# B&R Automation Studio project TD52 (part 123)

#### general_HCCyclic.st
```iecst
(*******************************************************************************
general_HC		general functions

This code is confidential and proprietary to the INNIO Company.
It may not be used in any form, or reproduced in any manner,
without the express written permission of the INNIO Company.
Copyright, INNIO Company, 2019

Customized modifications: -
------------------------

History:
-------
V0.00.0	25.04.2012	lettenb.	new
V3.99.0 21.02.2013	lettenb.	cleanup
V4.03.0 11.01.2015	Denk		Bugfix, OUT_HC.tHWF_Dem.Do not implemented
		15.03.2016	Denk		Bugfix, Handbedienebene. OR IN_HC.tManAuxCtr.bHWF_Dem;
V4.05.0 11.12.2017	lettenb.	check para setup added
V4.14.0 08.11.2024	Bacci		OUT_HC.tECW_ShutOffVal_Dem.Do, OUT_HC.tValHeater_Dem.Do, OUT_HC.tFanRingHeater_Dem.Do added

Instructions for use:
--------------------
Outstandings:
------------
*******************************************************************************)

PROGRAM _INIT

	xECW_ShutOffVal_Dem_Active.enable := TRUE;
	xECW_ShutOffVal_Dem_Active.pPVstring := ADR('HalIO::ECW_ShutOffVal_Dem');
	xECW_ShutOffVal_Dem_Active();
	bECW_ShutOffVal_Dem_Exist := xECW_ShutOffVal_Dem_Active.exist;

	xValHeater_Dem_Active.enable := TRUE;
	xValHeater_Dem_Active.pPVstring := ADR('HalIO::ValHeater_Dem');
	xValHeater_Dem_Active();
	bValHeater_Dem_Exist := xValHeater_Dem_Active.exist;

	xFanRingHeater_Dem_Active.enable := TRUE;
	xFanRingHeater_Dem_Active.pPVstring := ADR('HalIO::FanRingHeater_Dem');
	xFanRingHeater_Dem_Active();
	bFanRingHeater_Dem_Exist := xFanRingHeater_Dem_Active.exist;

END_PROGRAM

PROGRAM _CYCLIC

	(* check para setup *)
	IN_HC.tPB2MM.bParaSetupOk;
	Para.iEng_Motortype;    (* MIN= 208   MAX= 920    *)
	Para.rN_EngStart_LimHi; (* MIN= 50.0  MAX= 2200.0 *)

	(* engine type defnition *)
	xEngType.Motortype := INT_TO_UINT(Para.iEng_Motortype);
	xEngType();

	(* engine operating mode selection *)
	bOMSS_Stop := FALSE;
	bOMSS_Man  := FALSE;
	bOMSS_Aut  := FALSE;
	bOMSS_Test := FALSE;
	bOMSS_Scav := FALSE;
	bOMSS_MAT  := FALSE;

	CASE IN_HC.iIdx_OMSS OF
	0:	bOMSS_Stop := TRUE;
	1:	bOMSS_Man  := TRUE;
		bOMSS_MAT  := TRUE;
	2:	bOMSS_Aut  := TRUE;
		bOMSS_MAT  := TRUE;
	3:	bOMSS_Test := TRUE;
		bOMSS_MAT  := TRUE;
	4:	bOMSS_Scav := TRUE;
	END_CASE;

	(* engine operating mode *)
	xOpMode(in:= IN_HC.iSt_OpMode);

	(*----------------------------------------------------------------------------------*)
	(* engine start speed *)
	xGR_MAXR_N_EngStart(In:= IN_HC.rN_EngAct, Gw:= Para.rN_EngStart_LimHi, Hy:= Para.rN_EngStart_HyHi);
	xTOF_N_EngStart(IN:= xGR_MAXR_N_EngStart.Q AND IN_HC.tPB2MM.bParaSetupOk, PT:= T#10s);
	bN_EngStart := xTOF_N_EngStart.Q;

	(*----------------------------------------------------------------------------------*)
	(* demand heating circuit flap *)
	OUT_HC.tHWF_Dem.Do := (IN_HC.bEng_Aux_Dem_CDR AND NOT IN_HC.bMsg1053 AND NOT IN_HC.bMsg1054 AND NOT IN_HC.bMsg1031)
						   OR IN_HC.tManAuxCtr.bHWF_Dem;

	(*----------------------------------------------------------------------------------*)
	(* demand 2-way shut off valve engine jacket water circuit (P.04(06)-YCS-029) *)
	OUT_HC.tECW_ShutOffVal_Dem.Do := IN_HC.bEng_Aux_Dem_CDR;

	(*----------------------------------------------------------------------------------*)
	(* demand 3-way valve heater (P.04/06/07-H-001) *)
	OUT_HC.tValHeater_Dem.Do := (NOT bT_AirOutdoor_Hi1 AND Para.bT_AirOutdoor_Active)
							 	 AND NOT IN_HC.bMsg1031
								 AND NOT IN_HC.bMsg1053
								 AND NOT IN_HC.bMsg1054;

	(*----------------------------------------------------------------------------------*)
	(* demand fan ring heater (P.04/06/07/09H-100) *)
	OUT_HC.tFanRingHeater_Dem.Do := (NOT bT_AirOutdoor_Hi1 AND Para.bT_AirOutdoor_Active)
							 		 AND NOT IN_HC.bMsg1031
									 AND NOT IN_HC.bMsg1053
									 AND NOT IN_HC.bMsg1054;

END_PROGRAM
```

#### general_HC.var
```iecst
VAR
	xGR_MAXR_N_EngStart : GR_MAXR;
	xTOF_N_EngStart : TOF;
	xECW_ShutOffVal_Dem_Active : OutExist;
	xValHeater_Dem_Active : OutExist;
	xFanRingHeater_Dem_Active : OutExist;
END_VAR
```

### Program Logical/HeatingCooling/BHV (IEC, version 4.11.0) - boiler house ventilation

#### BHVCyclic.st
```iecst
(*******************************************************************************
BHV	Boiler house ventilation

This code is confidential AND proprietary to the INNIO Company.
It may NOT be used in any form, or reproduced in any manner,
without the express written permission of the INNIO Company.
Copyright, INNIO Company, 2022

Customized modifications: -
------------------------

History:
-------
V4.03.0	25.07.2015	Plattner Johannes
V4.11.0	17.01.2022	lettenb.	bFail_BHV: tBHV_Dem.Do added to avoid warning at standstill, bugfix

Instructions FOR use:
--------------------

Boiler house ventilation, activation AND demand

Outstandings:
------------
*******************************************************************************)
PROGRAM _CYCLIC

	(* boiler house ventilation aktive*)
	(*----------------------------------------------------------------------------*)
	IF Para.bBHV_Active THEN

		OUT_HC.tBHV_Dem.Do	:= (IN_HC.tDemnd_BHV.Di AND NOT IN_HC.tManAuxCtr.bBHV_Dem_Man)
							   OR IN_HC.tManAuxCtr.bBHV_Dem;	(* Manual operating auxiliaries control - Handbedienebene *)
		bFail_BHV		:= NOT IN_HC.tBHV_Op.Di AND OUT_HC.tBHV_Dem.Do;
		(*----------------------------------------------------------------------------*)

		(* boiler house ventilation inaktive*)
		(*----------------------------------------------------------------------------*)
	ELSE

		OUT_HC.tBHV_Dem.Do	:= FALSE;
		bFail_BHV			:= FALSE;

	END_IF;
	(*----------------------------------------------------------------------------*)

END_PROGRAM
```

### Program Logical/HeatingCooling/Pr_ECW (IEC, version 4.12.0) - pressure engine cooling water

#### Pr_ECWCyclic.st
```iecst
(*******************************************************************************
Pr_ECW			pressure engine cooling water

This code is confidential and proprietary to the INNIO Company.
It may not be used in any form, or reproduced in any manner,
without the express written permission of the INNIO Company.
Copyright, INNIO Company, 2023

Customized modifications: -
------------------------

History:
-------
V0.1	20.10.1998	Pa			erstellt
 		24.11.1998	Pa			Korrekturlesung
V1.80	06.03.2003	LH			VISU-Grenzwerte erst aktiv wenn Rezepte auf Steuerung sind
 		18.03.2003	LH			Einlesen Analogeingang --> pb17
V2.06	01.07.2004	LH			Messignalstörung mit 2mA verzögert
V2.07	03.09.2004	LH			getrennte Verzögerungen für Messignalstörung eingeführt
V1.90	29.03.2004	LH			GW Kühlwasserdruck minimum warnend (Abstellung + 0,2bar)
 								GW Kühlwasserdruck maximum warnend (Abstellung - 0,4bar)
V2.20	24.04.2007	LH			Filter: 200ms --> 500ms (Hirzinger)
V2.50.0 28.01.2009	lettenb.	calm: GW_KDMI_W, HY_KDMI_W new parameter
V3.30.0	15.12.2011	lettenb.	GW_KDMA_W = GW_KDMA - 20 (war 40) (anforderung christian lang)
V3.99.0 21.02.2013	lettenb.	kwd -> Pr_ECW renamed, cleaning
V4.04.0	25.10.2016	lettenb.	measuring signal plausibility check (Functional Safety EN 13849)
		03.02.2017				bTON_EngRun added (validation just for 1 time)
		21.02.2017				2763: 0,1 -> 0,01 bar(acc.spec.thummer)
V4.05.0	22.12.2017	lettenb.	comment added: Safety-related application software source code (EN 13849-1 / 4.6.3)
		31.01.2018				2763 new logic(false alarms after long engine stand still time)(gfoeller)
V4.11.0	05.11.2021	Schmid		new Pr_ECW plausibility check logic
V4.12.0	28.03.2023	Perktold	variant mech Pump: Pr_ECW paus. check 10s longer monitoring, pressure limit 15mbar (former 20mbar)
V4.14.0 10.12.2024	Nagy		Added bPr_ECW_LoLoPrio2, bPr_ECW_HiHiPrio2 (2024-225)
Instructions for use:
--------------------

Outstandings:
------------
(*******************************************************************************)

PROGRAM _CYCLIC

(*---------------------------------------------------------------------------*)
	(* engine cooling water pressure *)

	(* low *)
	xGRMIN_Pr_ECW_Lo(In:= IN_HC.tPr_ECW.Ai, Gw:= Para.rPr_ECW_LimLo, Hy:= Para.rPr_ECW_HyLo);
    xTON_Pr_ECW_Lo(IN:= xGRMIN_Pr_ECW_Lo.Q AND IN_HC.tPB2MM.bParaSetupOk AND IN_HC.tPr_ECW.GoodQual, PT:= T#20s);
    bPr_ECW_Lo := xTON_Pr_ECW_Lo.Q;
	(* low during operation*)
	xGRMIN_Pr_ECW_LimOp(In:= IN_HC.tPr_ECW.Ai, Gw:= Para.rPr_ECW_LimLo_EngOp, Hy:= Para.rPr_ECW_HyLo);
	xTON_Pr_ECW_LimOp(IN:= xGRMIN_Pr_ECW_LimOp.Q AND IN_HC.tPB2MM.bParaSetupOk AND IN_HC.tPr_ECW.GoodQual, PT:= T#20s);
	bPr_ECW_LimOp := xTON_Pr_ECW_LimOp.Q;
	(********************************************************************************************************************
	Safety-related application software source code (EN 13849-1 / 4.6.3): BEGIN
	*********************************************************************************************************************)
	(* low low *)
	xGRMIN_Pr_ECW_LoLo(In:= IN_HC.tPr_ECW.Ai, Gw:= Para.rPr_ECW_LimLoLo, Hy:= Para.rPr_ECW_HyLoLo);
    xTON_Pr_ECW_LoLo(IN:= xGRMIN_Pr_ECW_LoLo.Q AND IN_HC.tPB2MM.bParaSetupOk AND IN_HC.tPr_ECW.GoodQual, PT:= T#3s);
    bPr_ECW_LoLo := xTON_Pr_ECW_LoLo.Q;
	(********************************************************************************************************************
	Safety-related application software source code (EN 13849-1 / 4.6.3): END
	*********************************************************************************************************************)
	(* low low Prio2 *)
	xGRMIN_Pr_ECW_LoLoPrio2(In:= IN_HC.tPr_ECW.Ai, Gw:= Para.rPr_ECW_LimLoLo - 0.2);
	xTON_Pr_ECW_LoLoPrio2(IN:= xGRMIN_Pr_ECW_LoLoPrio2.Q AND IN_HC.tPB2MM.bParaSetupOk AND IN_HC.tPr_ECW.GoodQual, PT:= T#3s);
	bPr_ECW_LoLoPrio2 := xTON_Pr_ECW_LoLoPrio2.Q;

	(* low 1 *)(* for custom use *)
	xGRMIN_Pr_ECW_Lo1(In:= IN_HC.tPr_ECW.Ai, Gw:= Para.rPr_ECW_LimLo1, Hy:= Para.rPr_ECW_HyLo1);
    xTON_Pr_ECW_Lo1(IN:= xGRMIN_Pr_ECW_Lo1.Q AND IN_HC.tPB2MM.bParaSetupOk, PT:= T#3s);
    OUT_HC.bPr_ECW_Lo1 := xTON_Pr_ECW_Lo1.Q;

	(* high *)
	xGRMAX_Pr_ECW_Hi(In:= IN_HC.tPr_ECW.Ai, Gw:= Para.rPr_ECW_LimHiHi - 0.20, Hy:= Para.rPr_ECW_HyHiHi);
    xTON_Pr_ECW_Hi(IN:= xGRMAX_Pr_ECW_Hi.Q AND IN_HC.tPB2MM.bParaSetupOk, PT:= T#10s);
	bPr_ECW_Hi := xTON_Pr_ECW_Hi.Q;

	(* high high *)
	xGRMAX_Pr_ECW_HiHi(In:= IN_HC.tPr_ECW.Ai, Gw:= Para.rPr_ECW_LimHiHi, Hy:= Para.rPr_ECW_HyHiHi);
    xTON_Pr_ECW_HiHi(IN:= xGRMAX_Pr_ECW_HiHi.Q AND IN_HC.tPB2MM.bParaSetupOk, PT:= T#10s);
	bPr_ECW_HiHi := xTON_Pr_ECW_HiHi.Q;

	(* high high Prio2 *)
	xGRMAX_Pr_ECW_HiHiPrio2(In:= IN_HC.tPr_ECW.Ai, Gw:= Para.rPr_ECW_LimHiHi + 0.2);
	bPr_ECW_HiHiPrio2 := xGRMAX_Pr_ECW_HiHiPrio2.Q AND IN_HC.tPB2MM.bParaSetupOk;

	(********************************************************************************************************************
	Safety-related application software source code (EN 13849-1 / 4.6.3): BEGIN
	*********************************************************************************************************************)
	(* measuring signal plausibility check - engine cooling water pressure (Functional Safety) *)

	(* reset saved pressure values *)
	IF xF_TRIG_Pcheck_Meas.Q THEN
		rPr_ECW_MaxValue		:=	0.0;
		rPr_ECW_MinValue		:=	100.0;
	END_IF;

	(* determine point when ECWP starts *)
	rN_ThresSpeedUp		:=	900.0;
	rN_ThresEngStop		:=	5.0;
	IF IN_HC.bECWP_MechDriven THEN	xR_TRIG_ECWP_start.CLK	:=	(IN_HC.rN_EngAct > rN_ThresEngStop);	// problem of failed start attempt!
	ELSE							xR_TRIG_ECWP_start.CLK	:=	IN_HC.tECWP1Dem.Do;
	END_IF;
	xR_TRIG_ECWP_start();
	xTP_Pr_ECW_Min_ECWP_start(IN:= xR_TRIG_ECWP_start.Q, PT:= T#10s);
	IF NOT IN_HC.tECWP1Dem.Do THEN	xTP_Pr_ECW_Min_ECWP_start(IN:= FALSE, PT:= T#0s);
	END_IF;

	(* define time window for tracking minimum ECW pressure *)
	xTON_NEng_Exc_Thres(IN := (IN_HC.rN_EngAct > rN_ThresSpeedUp), PT := T#10s);								//10s delay after speed up rpm reached before monitoring stop
	xRS_Pr_ECW_Min_Meas.SET		:=	xR_TRIG_ECWP_start.Q;
	IF IN_HC.bECWP_MechDriven THEN	xRS_Pr_ECW_Min_Meas.RESET1	:=	xTON_NEng_Exc_Thres.Q						// speed up rpm reached + 10s TON
																OR	(IN_HC.rN_EngAct < rN_ThresEngStop);		// interrupt with failed start attempt
	ELSE							xRS_Pr_ECW_Min_Meas.RESET1	:=	NOT xTP_Pr_ECW_Min_ECWP_start.Q;
	END_IF;
	xRS_Pr_ECW_Min_Meas();

	(* determine minimum ECW pressure during time window *)
	IF xRS_Pr_ECW_Min_Meas.Q1 THEN
		IF (IN_HC.tPr_ECW.Ai < rPr_ECW_MinValue) THEN	rPr_ECW_MinValue	:=	IN_HC.tPr_ECW.Ai;
		END_IF;
		IF (IN_HC.tPr_ECW.Ai > rPr_ECW_MaxValue) THEN	rPr_ECW_MaxValue	:=	IN_HC.tPr_ECW.Ai;
		END_IF;
	END_IF;

	(* mute plausibility check after ECWP operation *)
	IF IN_HC.bECWP_MechDriven THEN	xTOF_Pcheck_MonDeact.IN	:=	(IN_HC.rN_EngAct > rN_ThresEngStop);		// delay w.r.t. engine coming to standstill
	ELSE							xTOF_Pcheck_MonDeact.IN	:=	IN_HC.tECWP1Dem.Do;
	END_IF;
	xTOF_Pcheck_MonDeact(PT:= T#60s);
	bPcheck_Pr_ECW_MonRel	:=	NOT (xTOF_Pcheck_MonDeact.Q AND NOT xTOF_Pcheck_MonDeact.IN)	// mute for fast ECWP or engine restart
							AND	IN_HC.bEng_Aux_Dem												// check only active when engine/auxiliaries demanded
							AND	IN_HC.tPB2MM.bParaSetupOk;										// scaling parameters for Pr_ECW loaded

	(* trigger check evaluation *)
	xF_TRIG_Pcheck_Meas(CLK:= xRS_Pr_ECW_Min_Meas.Q1);

	IF xF_TRIG_Pcheck_Meas.Q AND bPcheck_Pr_ECW_MonRel THEN		bPr_ECW_PcheckFail	:=	((rPr_ECW_MaxValue - rPr_ECW_MinValue) < 0.015);
	ELSE														bPr_ECW_PcheckFail	:=	FALSE;
	END_IF;

	IF MM2VIS.bMsg2104 OR NOT IN_HC.tECWP_Op.Di THEN						bPr_ECW_PcheckFail := FALSE;
	ELSIF (rPr_ECW_MaxValue = 0.0) THEN										bPr_ECW_PcheckFail := FALSE; (* value not valid *)
	ELSIF (rPr_ECW_MinValue  = 0.0) OR (rPr_ECW_MinValue  = 100.0) THEN		bPr_ECW_PcheckFail := FALSE; (* value not valid *)
	END_IF;
	(********************************************************************************************************************
	Safety-related application software source code (EN 13849-1 / 4.6.3): END
	*********************************************************************************************************************)

END_PROGRAM
```

#### Pr_ECW.var
```iecst
VAR
	xGRMIN_Pr_ECW_Lo : GR_MINR;
	xTON_Pr_ECW_Lo : TON;
	xGRMIN_Pr_ECW_LimOp : GR_MINR;
	xTON_Pr_ECW_LimOp : TON;
	xGRMIN_Pr_ECW_LoLo : GR_MINR;
	xTON_Pr_ECW_LoLo : TON;
	xTON_Pr_ECW_LoLoPrio2 : TON;
	xGRMIN_Pr_ECW_LoLoPrio2 : GR_MINR;
	xGRMIN_Pr_ECW_Lo1 : GR_MINR;
	xTON_Pr_ECW_Lo1 : TON;
	xGRMAX_Pr_ECW_Hi : GR_MAXR;
	xTON_Pr_ECW_Hi : TON;
	xGRMAX_Pr_ECW_HiHi : GR_MAXR;
	xGRMAX_Pr_ECW_HiHiPrio2 : GR_MAXR;
	xTON_Pr_ECW_HiHi : TON;
	xR_TRIG_ECWP_start : R_TRIG; (*v4.11 new Pr_ECW plausibility check*)
	xTP_Pr_ECW_Min_ECWP_start : TP; (*v4.11new Pr_ECW plausibility check*)
	xTOF_Pcheck_MonDeact : TOF; (*v4.11new Pr_ECW plausibility check*)
	xRS_Pr_ECW_Min_Meas : RS; (*v4.11 new Pr_ECW plausibility check*)
	xF_TRIG_Pcheck_Meas : F_TRIG; (*v4.11 new Pr_ECW plausibility check*)
	rN_ThresSpeedUp : REAL; (*v4.11 new Pr_ECW plausibility check*)
	rN_ThresEngStop : REAL; (*v4.11 new Pr_ECW plausibility check*)
	bPcheck_Pr_ECW_MonRel : BOOL; (*v4.11 new Pr_ECW plausibility check*)
	rPr_ECW_MinValue : REAL := 100.0; (*v4.11 new Pr_ECW plausibility check*)
	rPr_ECW_MaxValue : REAL := 0.0; (*v4.11 new Pr_ECW plausibility check*)
	xTON_NEng_Exc_Thres : TON;
END_VAR
```

### Program Logical/HeatingCooling/T_CD (IEC, version 4.03.0) - temperature condensor circuit

#### T_CDCyclic.st
```iecst
(*******************************************************************************
T_CD		temperature condensor circuit

This code is confidential and proprietary to the INNIO Company.
It may not be used in any form, or reproduced in any manner,
without the express written permission of the INNIO Company.
Copyright, INNIO Company, 2019

Customized modifications: -
------------------------

History:
-------
V4.03.0	27.07.2015	Plattner	task created

Instructions for use:
--------------------

Outstandings:
------------
*******************************************************************************)

PROGRAM _CYCLIC
	(*-----------------------------------------------------------------------------*)
	(* condensor circuit supply temperature *)
	(* high *)
	xGRMAX_T_CD_Su_Hi(Gw:= Para.rT_CD_Su_LimHi, Hy:= Para.rT_CD_Su_HyHi, In:= IN_HC.tT_CD_Su.Ai);
	xTON_T_CD_Su_Hi(IN:= xGRMAX_T_CD_Su_Hi.Q AND IN_HC.tPB2MM.bParaSetupOk AND Para.bT_CD_Su_Active, PT:= T#2s);
	bT_CD_Su_Hi := xTON_T_CD_Su_Hi.Q;

	(*-----------------------------------------------------------------------------*)
	(* condensor circuit temperature *)
	(* high *)
	xGRMAX_T_CD_Re_Hi(In:= IN_HC.tT_CD_Re.Ai, Gw:= Para.rT_CD_Re_LimHi, Hy:= Para.rT_CD_Re_HyHi);
	xTON_T_CD_Re_Hi(IN := xGRMAX_T_CD_Re_Hi.Q AND IN_HC.tPB2MM.bParaSetupOk AND Para.bT_CD_Re_Active, PT := T#2s);
	bT_CD_Re_Hi := xTON_T_CD_Re_Hi.Q;

	(*-----------------------------------------------------------------------------*)

END_PROGRAM
```

#### T_CD.var
```iecst
VAR
	xTON_T_CD_Su_Hi : TON;
	xGRMAX_T_CD_Su_Hi : GR_MAXR;
	xGRMAX_T_CD_Re_Hi : GR_MAXR;
	xTON_T_CD_Re_Hi : TON;
END_VAR
```

### Program Logical/HeatingCooling/T_ECW (IEC, version 4.00.0) - temperature engine cooling water

#### T_ECWCyclic.st
```iecst
(*******************************************************************************
T_ECW			temperature engine cooling water

This code is confidential and proprietary to the INNIO Company.
It may not be used in any form, or reproduced in any manner,
without the express written permission of the INNIO Company.
Copyright, INNIO Company, 2019

Customized modifications: -
------------------------

History:
-------
V0.1	01.10.1998	Pa			erstellt
		24.11.1998	Pa			korrekturlesung
V170	03.04.2002	LH			Verzögerung Kühlwassertemperatur max. => 5min
								Grenzwert Kühlwassertemperatur max. + 2°C (Abstellung)
V180	06.03.2003	LH			VISU-Grenzwerte erst aktiv wenn Rezepte auf Steuerung sind
		18.03.2003	LH			Einlesen Analogeingang --> pb17
V3.99.0	20.02.2013	lettenb.	kwtp renamed T_ECW, cleaning
								new param.for cooling water bypass valve
V4.00.0 19.03.2015				xGRMIN_T_ECW_Lo: avoid bMsg1145 at cold restart within hysteresis

Instructions for use:
--------------------

Outstandings:
------------
(*******************************************************************************)

PROGRAM _CYCLIC

(*---------------------------------------------------------------------------*)
	(* engine cooling water temperature *)

	(* low *)
	IF IN_HC.tPB2MM.bParaSetupOk THEN (* avoid bMsg1145 at cold restart within hysteresis *)
		 xGRMIN_T_ECW_Lo(In:= IN_HC.tT_ECW.Ai, Gw:= Para.rT_ECW_LimLo, Hy:= Para.rT_ECW_HyLo);
	ELSE xGRMIN_T_ECW_Lo(In:= 1.0, Gw:= 0.0, Hy:= 0.0);
	END_IF;
	xTON_T_ECW_Lo(IN:= xGRMIN_T_ECW_Lo.Q AND IN_HC.tPB2MM.bParaSetupOk, PT:= T#2s);
    OUT_HC.bT_ECW_Lo := xTON_T_ECW_Lo.Q;

	(*high preheating off *)
	xGRMAX_T_ECW_PreH_OFF(In:= IN_HC.tT_ECW.Ai, Gw:= Para.rT_ECW_PreH_LimOFF, Hy:= Para.rT_ECW_PreH_HyOFF);
    xTON_T_ECW_PreH_OFF(IN:= xGRMAX_T_ECW_PreH_OFF.Q AND IN_HC.tPB2MM.bParaSetupOk, PT:= T#2s);
    OUT_HC.bT_ECW_PreH_OFF := xTON_T_ECW_PreH_OFF.Q;

	(* high synch/load release *)
	xGRMAX_T_ECW_RelLoad(In:= IN_HC.tT_ECW.Ai, Gw:= Para.rT_ECW_LimRelLoad, Hy:= Para.rT_ECW_HyRelLoad);
    xTON_T_ECW_RelLoad(IN:= xGRMAX_T_ECW_RelLoad.Q AND IN_HC.tPB2MM.bParaSetupOk, PT:= T#2s);
    OUT_HC.bT_ECW_RelLoad := xTON_T_ECW_RelLoad.Q;

	(* high *)
	xGRMAX_T_ECW_Hi(In:= IN_HC.tT_ECW.Ai, Gw:= Para.rT_ECW_LimHi, Hy:= Para.rT_ECW_HyHi);
    xTON_T_ECW_Hi(IN:= xGRMAX_T_ECW_Hi.Q AND IN_HC.tPB2MM.bParaSetupOk, PT:= T#300s);
    OUT_HC.bT_ECW_Hi := xTON_T_ECW_Hi.Q;

	(* high high *)
	xGRMAX_T_ECW_HiHi(In:= IN_HC.tT_ECW.Ai, Gw:= Para.rT_ECW_LimHi + 2.0, Hy:= Para.rT_ECW_HyHi);
    xTON_T_ECW_HiHi(IN:= xGRMAX_T_ECW_HiHi.Q AND IN_HC.tPB2MM.bParaSetupOk, PT:= T#2s);
    bT_ECW_HiHi := xTON_T_ECW_HiHi.Q;

	(* high P2 *)
	xGRMAX_T_ECW_HiHiPrio2(In:= IN_HC.tT_ECW.Ai, Gw:= Para.rT_ECW_LimHi + 5.0, Hy:= Para.rT_ECW_HyHi);
	xTON_T_ECW_HiHiPrio2(IN:= xGRMAX_T_ECW_HiHiPrio2.Q AND IN_HC.tPB2MM.bParaSetupOk, PT:= T#2s);
	bT_ECW_HiHiPrio2 := xTON_T_ECW_HiHiPrio2.Q;

	(* high 1 *)
	xGRMAX_T_ECW_Hi1(In:= IN_HC.tT_ECW.Ai, Gw:= Para.rT_ECW_LimHi1, Hy:= Para.rT_ECW_HyHi1);
    xTON_T_ECW_Hi1(IN:= xGRMAX_T_ECW_Hi1.Q AND IN_HC.tPB2MM.bParaSetupOk, PT:= T#2s);
    bT_ECW_Hi1 := xTON_T_ECW_Hi1.Q;

	(* high 2 *)
	xGRMAX_T_ECW_Hi2(In:= IN_HC.tT_ECW.Ai, Gw:= Para.rT_ECW_LimHi2, Hy:= Para.rT_ECW_HyHi2);
    xTON_T_ECW_Hi2(IN:= xGRMAX_T_ECW_Hi2.Q AND IN_HC.tPB2MM.bParaSetupOk, PT:= T#2s);
    bT_ECW_Hi2 := xTON_T_ECW_Hi2.Q;

	(*---------------------------------------------------------------------------*)
	(* engine cooling water temperature - bypass valve *)
	xGRMIN_T_ECW_BpV(In:= IN_HC.tT_ECW.Ai, Gw:= Para.rT_ECW_LimBpV, Hy:= Para.rT_ECW_HyBpV);
	xTON_T_ECW_BpV(IN:= xGRMIN_T_ECW_BpV.Q, PT:= T#2s);

	bECW_DemBpV := (	IN_HC.bEng_Aux_Dem AND xTON_T_ECW_BpV.Q)
    			OR (NOT IN_HC.bEng_Aux_Dem AND IN_HC.bEng_Aux_Dem_CDR);
    OUT_HC.tECW_DemBpV.Do 	:= bECW_DemBpV;

	(*---------------------------------------------------------------------------*)
	(*	engine cooling water bypass pump *)
    bECW_DemBpP 			:= bECW_DemBpV;
    OUT_HC.tECW_DemBpP.Do 	:= bECW_DemBpP;

(*---------------------------------------------------------------------------*)

END_PROGRAM
```

#### T_ECW.var
```iecst
VAR
	xGRMIN_T_ECW_Lo : GR_MINR;
	xTON_T_ECW_Lo : TON;
	xGRMAX_T_ECW_PreH_OFF : GR_MAXR;
	xTON_T_ECW_PreH_OFF : TON;
	xGRMAX_T_ECW_RelLoad : GR_MAXR;
	xTON_T_ECW_RelLoad : TON;
	xGRMAX_T_ECW_Hi : GR_MAXR;
	xTON_T_ECW_Hi : TON;
	xGRMAX_T_ECW_HiHi : GR_MAXR;
	xTON_T_ECW_HiHi : TON;
	xGRMAX_T_ECW_HiHiPrio2 : GR_MAXR;
	xTON_T_ECW_HiHiPrio2 : TON;
	xGRMAX_T_ECW_Hi1 : GR_MAXR;
	xTON_T_ECW_Hi1 : TON;
	xGRMAX_T_ECW_Hi2 : GR_MAXR;
	xTON_T_ECW_Hi2 : TON;
	xGRMIN_T_ECW_BpV : GR_MINR;
	xTON_T_ECW_BpV : TON;
END_VAR
```

### Program Logical/HeatingCooling/T_EO (IEC, version 3.99.0) - temperature engine oil

#### T_EOCyclic.st
```iecst
(*******************************************************************************
T_EO			engine oil temperature

This code is confidential and proprietary to the INNIO Company.
It may not be used in any form, or reproduced in any manner,
without the express written permission of the INNIO Company.
Copyright, INNIO Company, 2019

Customized modifications: -
------------------------

History:
-------
V3.99.0	20.02.2013	lettenb.	new from task: otp

Instructions for use:
--------------------

Outstandings:
------------
(*******************************************************************************)

PROGRAM _CYCLIC

	(* engine oil temperature high 1 *)
	xGR_MAXR_T_EO_Hi1(In:= IN_HC.tT_EO.Ai, Gw:= Para.rT_EO_LimHi1, Hy:= Para.rT_EO_HyHi1);
	xTON_T_EO_Hi1(IN:= xGR_MAXR_T_EO_Hi1.Q AND IN_HC.tPB2MM.bParaSetupOk, PT:= T#2s);
	bT_EO_Hi1 := xTON_T_EO_Hi1.Q;

	(* engine oil temperature high 2 *)
	xGR_MAXR_T_EO_Hi2(In:= IN_HC.tT_EO.Ai, Gw:= Para.rT_EO_LimHi2, Hy:= Para.rT_EO_HyHi2);
	xTON_T_EO_Hi2(IN:= xGR_MAXR_T_EO_Hi2.Q AND IN_HC.tPB2MM.bParaSetupOk, PT:= T#2s);
	bT_EO_Hi2 := xTON_T_EO_Hi2.Q;

END_PROGRAM
```

#### T_EO.var
```iecst
VAR
	xTON_T_EO_Hi1 : TON;
	xGR_MAXR_T_EO_Hi1 : GR_MAXR;
	xTON_T_EO_Hi2 : TON;
	xGR_MAXR_T_EO_Hi2 : GR_MAXR;
END_VAR
```

### Program Logical/HeatingCooling/T_HW (IEC, version 4.05.0) - temperature heat water

#### T_HWCyclic.st
```iecst
(*******************************************************************************
T_HW		temperature heat water

This code is confidential and proprietary to the INNIO Company.
It may not be used in any form, or reproduced in any manner,
without the express written permission of the INNIO Company.
Copyright, INNIO Company, 2019

Customized modifications: -
------------------------

History:
-------
V3.99.0	20.02.2013	lettenb.	from task vltp, rltp, rltp_nk, rlt_m
								p_limitHC included
		14.03.2012	lettenb.	p_lim --> p_red (power red.from act.frozen power value) request: systems/thummer mathias
V4.00.0	01.07.2014	lettenb.	bT_HW_Su_Hi/HiHi: AND Para.bT_HW_Su_Active added, bugfix
V4.03.0	29.07.2015	plattner	heat circuit temperature added
V4.04.0 29.07.2016	lettenb.	2nd bT_HW_ReBeEng_Hi building removed, cleanup
		12.09.2016				comment removed
V4.05.0 13.06.2017	lettenb.	rP_Red_T_ECW_Low_Norm added, SWAT920/3

Instructions for use:
--------------------

Outstandings:
------------
*******************************************************************************)

PROGRAM _CYCLIC
	(*-----------------------------------------------------------------------------*)
	(* heat water supply temperature *)
	(* high *) (* W2430 *)
	xGRMAX_T_HW_Su_Hi(Gw:= Para.rT_HW_Su_LimHi, Hy:= Para.rT_HW_Su_HyHi, In:= IN_HC.tT_HW_Su.Ai);
	xTON_T_HW_Su_Hi(IN:= xGRMAX_T_HW_Su_Hi.Q AND IN_HC.tPB2MM.bParaSetupOk AND Para.bT_HW_Su_Active, PT:= T#2s);
	bT_HW_Su_Hi := xTON_T_HW_Su_Hi.Q;

	(* high high *) (* A1063 *)
	xGRMAX_T_HW_Su_HiHi(Gw:= Para.rT_HW_Su_LimHiHi, Hy:= Para.rT_HW_Su_HyHiHi, In:= IN_HC.tT_HW_Su.Ai);
	xTON_T_HW_Su_HiHi(IN := xGRMAX_T_HW_Su_HiHi.Q AND IN_HC.tPB2MM.bParaSetupOk AND Para.bT_HW_Su_Active, PT := T#2s);
	bT_HW_Su_HiHi := xTON_T_HW_Su_HiHi.Q;

	(*-----------------------------------------------------------------------------*)
	(* heat water return temperature *)
	(* high *)
	xGRMAX_T_HW_Re_Hi(In:= IN_HC.tT_HW_Re.Ai, Gw:= Para.rT_HW_Re_LimHi, Hy:= Para.rT_HW_Re_HyHi);
	xTON_T_HW_Re_Hi(IN := xGRMAX_T_HW_Re_Hi.Q AND IN_HC.tPB2MM.bParaSetupOk AND Para.bT_HW_Re_Active, PT := T#2s);
	bT_HW_Re_Hi := xTON_T_HW_Re_Hi.Q;

	(* high high *)
	xGRMAX_T_HW_Re_HiHi(In := IN_HC.tT_HW_Re.Ai, Gw := Para.rT_HW_Re_LimHiHi, Hy := Para.rT_HW_Re_HyHiHi);
	xTON_T_HW_Re_HiHi(IN:= xGRMAX_T_HW_Re_HiHi.Q AND IN_HC.tPB2MM.bParaSetupOk AND Para.bT_HW_Re_Active, PT:= T#2s);
	bT_HW_Re_HiHi := xTON_T_HW_Re_HiHi.Q;

	(*-----------------------------------------------------------------------------*)
	(* heat water return temperature after emergency cooler *)
	(* high *)
	xGRMAX_T_HW_ReAfEC_Hi(In:= IN_HC.tT_HW_ReAfEC.Ai, Gw:= Para.rT_HW_ReAfEC_LimHi, Hy:= Para.rT_HW_ReAfEC_HyHi);
	xTON_T_HW_ReAfEC_Hi(IN:= xGRMAX_T_HW_ReAfEC_Hi.Q AND IN_HC.tPB2MM.bParaSetupOk, PT:= T#2s);
	bT_HW_ReAfEC_Hi := xTON_T_HW_ReAfEC_Hi.Q;

	(* high high *)
	xGRMAX_T_HW_ReAfEC_HiHi(In:= IN_HC.tT_HW_ReAfEC.Ai, Gw:= Para.rT_HW_ReAfEC_LimHiHi, Hy:= Para.rT_HW_ReAfEC_HyHiHi);
	xTON_T_HW_ReAfEC_HiHi(IN:= xGRMAX_T_HW_ReAfEC_HiHi.Q AND IN_HC.tPB2MM.bParaSetupOk, PT:= T#2s);
	bT_HW_ReAfEC_HiHi := xTON_T_HW_ReAfEC_HiHi.Q;

	(*-----------------------------------------------------------------------------*)
	(* heat water return temperature before engine *)
	(* high *)
	xGRMAX_T_HW_ReBeEng_Hi(In:= IN_HC.tT_HW_ReBeEng.Ai, Gw:= Para.rT_HW_ReBeEng_LimHi, Hy:= Para.rT_HW_ReBeEng_HyHi, );
	xTON_T_HW_ReBeEng_Hi(IN:= xGRMAX_T_HW_ReBeEng_Hi.Q AND IN_HC.tPB2MM.bParaSetupOk, PT:= T#2s);
	bT_HW_ReBeEng_Hi := xTON_T_HW_ReBeEng_Hi.Q;

	(* high high *)(* reserve *)
	xGRMAX_T_HW_ReBeEng_HiHi(In:= IN_HC.tT_HW_ReBeEng.Ai, Gw:= Para.rT_HW_ReBeEng_LimHiHi, Hy:= Para.rT_HW_ReBeEng_HyHiHi, );
	xTON_T_HW_ReBeEng_HiHi(IN:= xGRMAX_T_HW_ReBeEng_HiHi.Q AND IN_HC.tPB2MM.bParaSetupOk, PT:= T#2s);
	bT_HW_ReBeEng_HiHi := xTON_T_HW_ReBeEng_HiHi.Q;

	(*-----------------------------------------------------------------------------*)
	(* heat circuit temperature *)
	(* high *)
	xGRMAX_T_HW_HC_Re_Hi(Gw:= Para.rT_HW_HC_Re_LimHi, Hy:= Para.rT_HW_HC_Re_HyHi, In:= IN_HC.tT_HW_HC_Re.Ai);
	xTON_T_HW_HC_Re_Hi(IN:= xGRMAX_T_HW_HC_Re_Hi.Q AND IN_HC.tPB2MM.bParaSetupOk AND Para.bT_HW_HC_Re_Active, PT:= T#2s);
	bT_HW_HC_Re_Hi := xTON_T_HW_HC_Re_Hi.Q;

	(*-----------------------------------------------------------------------------*)
	(* power reduction by heat water return temperature high *)
	(* selection *)
	CASE Para.iPred_T_HW_Re_Sel OF
		0:	rT_HW_Re := 0;						(* disabled	*)
		1:	rT_HW_Re := IN_HC.tT_HW_Re.Ai;		(* P.06(04)-TI-012	(NUT12) *)
		2:	rT_HW_Re := IN_HC.tT_HW_ReAfEC.Ai;	(* P.06(04)-TI-015	(NUT15) *)
		3:	rT_HW_Re := IN_HC.tT_HW_ReBeEng.Ai;	(* M.06(04)-TI-001	(NUT56) *)
		ELSE
			rT_HW_Re :=0;
	END_CASE;

	IF rT_HW_Re <= Para.rT_Pred_HW_Re_Start THEN
		rP_Act_Norm_frozen := IN_HC.rP_Act_Norm_Filt;
	END_IF;

	IF Para.iPred_T_HW_Re_Sel <> 0 AND rT_HW_Re > Para.rT_Pred_HW_Re_Start THEN
		OUT_HC.rP_Red_T_HWR_Norm := LIMIT(0.5, rP_Act_Norm_frozen - ((rT_HW_Re - Para.rT_Pred_HW_Re_Start) * Para.rPred_T_HW_Re_Rate), 1.0);
	ELSE
		OUT_HC.rP_Red_T_HWR_Norm := 1.0;
	END_IF;

	(* power reduction by engine cooling water return temperature low - warm up operation *)
	IF IN_HC.tT_ECW.Ai < Para.rT_ECW_PwrRamp_LimLo AND bOMSS_Man AND xEngType.Type9 THEN
		OUT_HC.rP_Red_T_ECW_Low_Norm := 0.40;//%Pnom(10MW) = ca.4MW
	ELSE
		OUT_HC.rP_Red_T_ECW_Low_Norm := 1.0;
	END_IF;

	(* power reduction by engine cooling water temperature high *)
	OUT_HC.rP_Red_T_ECW_Norm := LIMIT(0.5, 1.0 - ((IN_HC.tT_ECW.Ai - Para.rT_Pred_ECW_Start) * Para.rPred_ECW_Rate), 1.0);

	(*-----------------------------------------------------------------------------*)

	(*-----------------------------------------------------------------------------*)

END_PROGRAM
```

#### T_HW.var
```iecst
VAR
	xGRMAX_T_HW_Su_Hi : GR_MAXR;
	xTON_T_HW_Su_Hi : TON;
	xGRMAX_T_HW_Su_HiHi : GR_MAXR;
	xTON_T_HW_Su_HiHi : TON;
	xGRMAX_T_HW_Re_Hi : GR_MAXR;
	xTON_T_HW_Re_Hi : TON;
	xGRMAX_T_HW_Re_HiHi : GR_MAXR;
	xTON_T_HW_Re_HiHi : TON;
	xGRMAX_T_HW_ReBeEng_Hi : GR_MAXR;
	xTON_T_HW_ReBeEng_Hi : TON;
	xGRMAX_T_HW_ReBeEng_HiHi : GR_MAXR;
	xTON_T_HW_ReBeEng_HiHi : TON;
	xGRMAX_T_HW_ReAfEC_Hi : GR_MAXR;
	xTON_T_HW_ReAfEC_Hi : TON;
	xGRMAX_T_HW_ReAfEC_HiHi : GR_MAXR;
	xTON_T_HW_ReAfEC_HiHi : TON;
	rT_HW_Re : REAL;
	rP_Act_Norm_frozen : REAL;
	xGRMAX_T_HW_HC_Re_Hi : GR_MAXR;
	xTON_T_HW_HC_Re_Hi : TON;
END_VAR
```

### Program Logical/HeatingCooling/T_AirOutdoor (IEC, version 3.99.0) - temperature air outdoor

#### T_AirOutdoor.st
```iecst
(*******************************************************************************
T_AirOutdoor		temperature air outdoor

This code is confidential and proprietary to the INNIO Company.
It may not be used in any form, or reproduced in any manner,
without the express written permission of the INNIO Company.
Copyright, INNIO Company, 2019

Customized modifications: -
------------------------

History:
-------
V2.10	18.05.2004	LH			erstellt
V3.99.0	21.02.2013	lettenb.	ult --> T_AirOutdoor renamed

Instructions for use:
--------------------

Outstandings:
------------
*******************************************************************************)

PROGRAM _CYCLIC

	(* outdoor air temperature *)

	(* high 1 *)
	xGRMAX_T_AirOutdoor_Hi1(In:= IN_HC.tT_AirOutdoor.Ai, Gw:= Para.rT_AirOutdoor_LimHi1, Hy:= Para.rT_AirOutdoor_HyHi1);
	bT_AirOutdoor_Hi1 := IN_HC.tPB2MM.bParaSetupOk AND xGRMAX_T_AirOutdoor_Hi1.Q AND Para.bT_AirOutdoor_Active;

	(* high 2 *)
	xGRMAX_T_AirOutdoor_Hi2(In:= IN_HC.tT_AirOutdoor.Ai, Gw:= Para.rT_AirOutdoor_LimHi2, Hy:= Para.rT_AirOutdoor_HyHi2);
	bT_AirOutdoor_Hi2 := IN_HC.tPB2MM.bParaSetupOk AND xGRMAX_T_AirOutdoor_Hi2.Q AND Para.bT_AirOutdoor_Active;

	(* high 3 *)
	xGRMAX_T_AirOutdoor_Hi3(In:= IN_HC.tT_AirOutdoor.Ai, Gw:= Para.rT_AirOutdoor_LimHi3, Hy:= Para.rT_AirOutdoor_HyHi3);
	bT_AirOutdoor_Hi3 := IN_HC.tPB2MM.bParaSetupOk AND xGRMAX_T_AirOutdoor_Hi3.Q AND Para.bT_AirOutdoor_Active;

	(* high 4 *)
	xGRMAX_T_AirOutdoor_Hi4(In:= IN_HC.tT_AirOutdoor.Ai, Gw:= Para.rT_AirOutdoor_LimHi4, Hy:= Para.rT_AirOutdoor_HyHi4);
	bT_AirOutdoor_Hi4 := IN_HC.tPB2MM.bParaSetupOk AND xGRMAX_T_AirOutdoor_Hi4.Q AND Para.bT_AirOutdoor_Active;

END_PROGRAM
```

#### T_AirOutdoor.var
```iecst
VAR
	xGRMAX_T_AirOutdoor_Hi1 : GR_MAXR;
	xGRMAX_T_AirOutdoor_Hi2 : GR_MAXR;
	xGRMAX_T_AirOutdoor_Hi3 : GR_MAXR;
	xGRMAX_T_AirOutdoor_Hi4 : GR_MAXR;
END_VAR
```

### Program Logical/HeatingCooling/T_Ch (IEC, version 4.07.0) - temperature charge air/mixture

#### T_ChCyclic.st
```iecst
(*******************************************************************************
T_Ch 		temperature charge air/mixture

This code is confidential and proprietary to the INNIO Company.
It may not be used in any form, or reproduced in any manner,
without the express written permission of the INNIO Company.
Copyright, INNIO Company, 2019

Customized modifications: -
------------------------

History:
-------
V3.99.0	21.02.2013	lettenb.	new for MM_HC
V4.07.0	09.08.2018	Schmid		2nd low temperature charge cooling circuit added

Instructions for use:
--------------------

Outstandings:
------------
*******************************************************************************)

PROGRAM _CYCLIC

	(* charge temperature t2' *)
	(* high 1 *)
	xGRMAX_T_Ch_Hi1(In:= IN_HC.rT_Ch_T2s_Avg, Gw:= Para.rT_Ch_LimHi1, Hy:= Para.rT_Ch_HyHi1);
	bT_Ch_Hi1 := xGRMAX_T_Ch_Hi1.Q AND IN_HC.tPB2MM.bParaSetupOk;

	(* high 2 *)
	xGRMAX_T_Ch_Hi2(In:= IN_HC.rT_Ch_T2s_Avg, Gw:= Para.rT_Ch_LimHi2, Hy:= Para.rT_Ch_HyHi2);
	bT_Ch_Hi2 := xGRMAX_T_Ch_Hi2.Q AND IN_HC.tPB2MM.bParaSetupOk;

	(* charge temperature before high-pressure turbo charger T1-HP - 2nd LT cooling circuit*)
	(* high 1 *)
	xGRMAX_T_Ch_T1HP_Hi1(In:= IN_HC.rT_Ch_T1HP_Avg, Gw:= Para.rT_Ch_T1HP_LimHi1, Hy:= Para.rT_Ch_T1HP_HyHi1);
	bT_Ch2_Hi1 := xGRMAX_T_Ch_T1HP_Hi1.Q AND IN_HC.tPB2MM.bParaSetupOk;

	(* high 2 *)
	xGRMAX_T_Ch_T1HP_Hi2(In:= IN_HC.rT_Ch_T1HP_Avg, Gw:= Para.rT_Ch_T1HP_LimHi2, Hy:= Para.rT_Ch_T1HP_HyHi2);
	bT_Ch2_Hi2 := xGRMAX_T_Ch_T1HP_Hi2.Q AND IN_HC.tPB2MM.bParaSetupOk;

END_PROGRAM
```

#### T_Ch.var
```iecst
VAR
	xGRMAX_T_Ch_Hi1 : GR_MAXR;
	xGRMAX_T_Ch_Hi2 : GR_MAXR;
	xGRMAX_T_Ch_T1HP_Hi1 : GR_MAXR;
	xGRMAX_T_Ch_T1HP_Hi2 : GR_MAXR;
END_VAR
```

### Program Logical/HeatingCooling/EC_Seq (IEC, version 4.03.0) - emergency cooler sequence

#### EC_SeqCyclic.st
```iecst
(*******************************************************************************
EC_Seq 			emergency cooler - sequence for 16 stages

This code is confidential and proprietary to the INNIO Company.
It may not be used in any form, or reproduced in any manner,
without written permission of the INNIO Company.
Copyright, INNIO Company, 2019

Customized modifications: -
------------------------

History:
-------
V0.1 	31-01-2003	Thaler		generated
     	21-03-2003	Thaler		last modification
V1.81	16-06-2003	LH			bits für Anzeige auf VISU
V1.82	16-09-2003	LH			Variable für XT-Anzeige
V2.07.1a31-03-2005	LH			Variable für Freigabe XT-Anzeige
V2.30	24-01-2008	LH			Variable für Freigabe XT-Anzeige gelöscht (Parameter!)
V3.99.0	21.02.2013	lettenb.	kv_seq -> EC_Seq renamed
V4.03.0 07.08.2015  Denk		Manual operating auxiliaries control functionality added

Instructions for use:
--------------------

Outstandings:
------------
*******************************************************************************)
PROGRAM _CYCLIC

	(* Manual operating auxiliaries control - Handbedienebene *)
	K_Var := LIMIT(0, Para.iEC_OpMode, 3);
	FOR i:= 1 TO Para.iEC_NumStages BY 1 DO
		IF 	(K_Var > 0 AND K_Var < 4) THEN
			K_ST1_ManAuxCtr  := IN_HC.tManAuxCtr.bEC_DemFan;
			K_ST2_ManAuxCtr  :=	IN_HC.tManAuxCtr.bEC_DemFan;
			K_ST3_ManAuxCtr  :=	IN_HC.tManAuxCtr.bEC_DemFan;
			K_ST4_ManAuxCtr  := IN_HC.tManAuxCtr.bEC_DemFan;
			K_ST5_ManAuxCtr  := IN_HC.tManAuxCtr.bEC_DemFan;
			K_ST6_ManAuxCtr  := IN_HC.tManAuxCtr.bEC_DemFan;
			K_ST7_ManAuxCtr  := IN_HC.tManAuxCtr.bEC_DemFan;
			K_ST8_ManAuxCtr  := IN_HC.tManAuxCtr.bEC_DemFan;
			K_ST9_ManAuxCtr  := IN_HC.tManAuxCtr.bEC_DemFan;
			K_ST10_ManAuxCtr := IN_HC.tManAuxCtr.bEC_DemFan;
			K_ST11_ManAuxCtr := IN_HC.tManAuxCtr.bEC_DemFan;
			K_ST12_ManAuxCtr := IN_HC.tManAuxCtr.bEC_DemFan;
			K_ST13_ManAuxCtr := IN_HC.tManAuxCtr.bEC_DemFan;
			K_ST14_ManAuxCtr := IN_HC.tManAuxCtr.bEC_DemFan;
			K_ST15_ManAuxCtr := IN_HC.tManAuxCtr.bEC_DemFan;
			K_ST16_ManAuxCtr := IN_HC.tManAuxCtr.bEC_DemFan;

			IF IN_HC.tManAuxCtr.bEC_DemFan = TRUE THEN
				iSumEC_Stages_ManAuxCtr := Para.iEC_NumStages;
			ELSE
				iSumEC_Stages_ManAuxCtr := 0;
			END_IF;
		END_IF;
	END_FOR;

	(* connection of in-/outputs *)
	EN[1]  := K_ST_1;
	EN[2]  := K_ST_2;
	EN[3]  := K_ST_3;
	EN[4]  := K_ST_4;
	EN[5]  := K_ST_5;
	EN[6]  := K_ST_6;
	EN[7]  := K_ST_7;
	EN[8]  := K_ST_8;
	EN[9]  := K_ST_9;
	EN[10] := K_ST_10;
	EN[11] := K_ST_11;
	EN[12] := K_ST_12;
	EN[13] := K_ST_13;
	EN[14] := K_ST_14;
	EN[15] := K_ST_15;
	EN[16] := K_ST_16;

	IN[1]  := K_ST1;
	IN[2]  := K_ST2;
	IN[3]  := K_ST3;
	IN[4]  := K_ST4;
	IN[5]  := K_ST5;
	IN[6]  := K_ST6;
	IN[7]  := K_ST7;
	IN[8]  := K_ST8;
	IN[9]  := K_ST9;
	IN[10] := K_ST10;
	IN[11] := K_ST11;
	IN[12] := K_ST12;
	IN[13] := K_ST13;
	IN[14] := K_ST14;
	IN[15] := K_ST15;
	IN[16] := K_ST16;

	OUT_HC.tEC_DemFan1.Do := Q[1] OR K_ST1_ManAuxCtr;
	OUT_HC.tEC_DemFan2.Do := Q[2] OR K_ST2_ManAuxCtr;
	OUT_HC.tEC_DemFan3.Do := Q[3] OR K_ST3_ManAuxCtr;
	OUT_HC.tEC_DemFan4.Do := Q[4] OR K_ST4_ManAuxCtr;
	OUT_HC.tEC_DemFan5.Do := Q[5] OR K_ST5_ManAuxCtr;
	OUT_HC.tEC_DemFan6.Do := Q[6] OR K_ST6_ManAuxCtr;
	OUT_HC.tEC_DemFan7.Do := Q[7] OR K_ST7_ManAuxCtr;
	OUT_HC.tEC_DemFan8.Do := Q[8] OR K_ST8_ManAuxCtr;
	OUT_HC.tEC_DemFan9.Do := Q[9] OR K_ST9_ManAuxCtr;
	OUT_HC.tEC_DemFan10.Do := Q[10] OR K_ST10_ManAuxCtr;
	OUT_HC.tEC_DemFan11.Do := Q[11] OR K_ST11_ManAuxCtr;
	OUT_HC.tEC_DemFan12.Do := Q[12] OR K_ST12_ManAuxCtr;
	OUT_HC.tEC_DemFan13.Do := Q[13] OR K_ST13_ManAuxCtr;
	OUT_HC.tEC_DemFan14.Do := Q[14] OR K_ST14_ManAuxCtr;
	OUT_HC.tEC_DemFan15.Do := Q[15] OR K_ST15_ManAuxCtr;
	OUT_HC.tEC_DemFan16.Do := Q[16] OR K_ST16_ManAuxCtr;

	(******************************************************************************)

	and_16b   (ADR(EN), ADR(Q), ADR(Q));	(* switch off "Q" if "EN" is FALSE:	"Q" := "EN" AND "Q" *)
	andnt_16b (ADR(EN), ADR(Q), ADR(RDY));	(* enabled outputs with status FALSE: "RDY" := "EN" AND NOT "Q" *)

	(* SEQU_C = stage number for stage numbers > iPriorityStage *)
	FOR i := (iPriorityStage + 1) TO 16 BY 1 DO
		SEQU_C[i] := i;
	END_FOR;

	(* SEQU_C = stage number + 100 for stage numbers <= iPriorityStage *)
	FOR i := iPriorityStage TO 1 BY -1 DO
		 SEQU_C[i] := i + 100;
	END_FOR;

	min_16di (ADR(RDY), ADR(SEQU_C), ADR(NEXT_ON));	(* stage for next on  as BOOL *)
	min_16di (ADR(Q), ADR(SEQU_C), ADR(NEXT_OFF)); 	(* stage for next off as BOOL *)

	iNextOn   := max_i_16b (ADR(NEXT_ON)); 			(* stage for next on  as INT  *)
	iNextOff  := max_i_16b (ADR(NEXT_OFF));			(* stage for next off as INT  *)

	iIN := max_i_16b (ADR(IN));						(* input : number of stages as INT *)
	iQ  := sum_16b (ADR(Q));   						(* output: number of stages as INT *)

	IF (iIN > iQ) THEN
		Q[iNextOn] := TRUE;
		iPriorityStage := iNextOn;
	END_IF;

	IF (iIN < iQ) THEN
		Q[iNextOff] := FALSE;
	END_IF;

	(******************************************************************************)

	(* bits for visu *)
	summe := 0;
	FOR i:= 1 TO 16 BY 1 DO
		summe := summe + Q[i];
	END_FOR;

	K_byte1	:= FALSE;
	K_byte2	:= FALSE;

	K_bit10	:= FALSE;
	K_bit11	:= FALSE;
	K_bit12	:= FALSE;

	K_bit20	:= FALSE;
	K_bit21	:= FALSE;
	K_bit22	:= FALSE;

	IF	(summe > 0) AND (summe < 9) THEN
		K_byte1	:= TRUE;
	END_IF;

	IF	((summe = 2) OR (summe = 4) OR (summe = 6) OR (summe = 8)) THEN
		K_bit10	:= TRUE;
	END_IF;

	IF	((summe = 3) OR (summe = 4) OR (summe = 7) OR (summe = 8)) THEN
		K_bit11	:= TRUE;
	END_IF;

	IF	((summe = 5) OR (summe = 6) OR (summe = 7) OR (summe = 8)) THEN
		K_bit12	:= TRUE;
	END_IF;

	IF	(summe > 8) THEN
		K_byte2	:= TRUE;
	END_IF;

	IF	((summe = 10) OR (summe = 12) OR (summe = 14) OR (summe = 16)) THEN
		K_bit20	:= TRUE;
	END_IF;

	IF	((summe = 11) OR (summe = 12) OR (summe = 15) OR (summe = 16)) THEN
		K_bit21	:= TRUE;
	END_IF;

	IF	((summe = 13) OR (summe = 14) OR (summe = 15) OR (summe = 16)) THEN
		K_bit22	:= TRUE;
	END_IF;

	IF iSumEC_Stages_ManAuxCtr > 0 THEN
		iSumEC_Stages := iSumEC_Stages_ManAuxCtr; 	(* Manual operating auxiliaries control - Handbedienebene to vis *)
	ELSE
		iSumEC_Stages := summe;						(* to vis *)
	END_IF;

END_PROGRAM
```

#### EC_Seq.var
```iecst
VAR
	K_bit10 : BOOL := 0; (* Kühlerstufe 1-8 bit0 *)
	K_bit11 : BOOL := 0; (* Kühlerstufe 1-8 bit1 *)
	K_bit12 : BOOL := 0; (* Kühlerstufe 1-8 bit2 *)
	K_bit20 : BOOL := 0; (* Kühlerstufe 9-16 bit0 *)
	K_bit21 : BOOL := 0; (* Kühlerstufe 9-16 bit1 *)
	K_bit22 : BOOL := 0; (* Kühlerstufe 9-16 bit2 *)
	K_byte1 : BOOL := 0; (* Kühlerstufen 1-8 *)
	K_byte2 : BOOL := 0; (* Kühlerstufen 9-16 *)
	IN : ARRAY[0..16] OF BOOL;
	Q : ARRAY[0..16] OF BOOL;
	RDY : ARRAY[0..16] OF BOOL;
	EN : ARRAY[0..16] OF BOOL;
	iQ : INT;
	iIN : INT;
	iPriorityStage : INT;
	SEQU_C : ARRAY[0..16] OF DINT;
	NEXT_ON : ARRAY[0..16] OF BOOL;
	NEXT_OFF : ARRAY[0..16] OF BOOL;
	i : INT;
	iNextOn : INT;
	iNextOff : INT;
	summe : USINT := 0;
	K_Var : INT; (*emergency cooler variant*)
	iSumEC_Stages_ManAuxCtr : INT; (*summary emergency cooler stages from Manual operating auxiliaries control *)
END_VAR
```

### Program Logical/HeatingCooling/EC (IEC, version 4.10.0) - emergency cooler

#### ECCyclic.st
```iecst
(*******************************************************************************
EC 			emergency cooler

This code is confidential and proprietary to the INNIO Company.
It may not be used in any form, or reproduced in any manner,
without written permission of the INNIO Company.
Copyright, INNIO Company, 2021

Customized modifications: -
------------------------

History:
-------
V0.1	03.07.1998	Pa			erstellt
 		24.11.1998	Pa			korrekturlesung
V172	20.08.2002	LH			überarbeitet
V173	27.09.2002	LH			Fehler in Abschaltung Stufe 7 korrigiert
V180	25.02.2003	LH			nkv_schr --> kv_schr, Ausgangsvariablen umbenannt, Grenzwerte über Rezept
		07.03.2003	LH			Freigabe Kühler umgebaut für Service
V181	05.06.2003	LH			Kontaktplan --> strukturierten Text
V183	16.09.2003	LH			Korrektur Vorzeichen P-Anteil
		12.12.2003	LH			Variante Kombikühler
V2071	03.01.2005	LH			Korrektur Start Kühler durch Temperaturgrenzwerte,
								Ansteuerung Notkühlpumpe nur über Ventilstellung
V2071b	28.06.2005	LH			Korrektur Start Kühler über Ventilstellung
V190	08.09.2004	LH			Erweiterung auf 11 Regler für XT
V2102	22.11.2006	LH			Korrektur Ansteuerung Notkühlpumpe für ausgebundenen Notkühlkreis und Kombikühler
V230	24.01.2008	LH			Abarbeitung nur wenn Kühler vorhanden ist (Para.iEC_OpMode <> 0)
		06.02.2008	LH			angepasst an Auto-Tune Regler
V2.34.0 23.10.2008	lettenb.	OUT_HC.bEC_Stage1-16:(FA_K_EIN.Q OR Kombi_K) added(fan only if OUT_HC.bEC_DemP)
V3.10.0 17.02.2010	lettenb. 	corr.demand fan stage 1,2 (brackets)	fehlerbehebung(robert mayer)
V3.20.0	11.11.2010	lettenb. 	Anz_anfhbt, K_Var, K_Anz, K_reg -> parameters
V3.99.0	21.02.2013	lettenb.	parts from pb3 included
		24.06.2013				GRMin_Ventpos2,xGRMax_Ventpos2,GRMax_Ventpos4: Hy:= 1->0.01, bugfix
V4.00.0	03.03.2015	lettenb.	K_frg (IN_HC.bEC_Rel) moved to MM_CU
V4.03.0 07.08.2015  Denk		Manual operating auxiliaries control functionality added
V4.07.0	08.01.2019	Schmid		redundant pump control
V4.10.0	02.02.2021	lettenb.	OUT_HC.tEC_DemPump.Do only when	auxiliaries demanded(bEng_Aux_Dem_CDR)
								for safety purposes: otherwise pump starts immediately when y-limit is reached(or setted manually)
								OUT_HC.bEmCWP_Dem for K_Var > 0 prepared for reduntant pumps, bugfix

Instructions for use:
--------------------

Outstandings:
------------
(*******************************************************************************)
PROGRAM _CYCLIC

	(*------------------------------------------------------------------------------------------*)
	(* parameters *)
	K_Var 		:= 				LIMIT(0, Para.iEC_OpMode, 3);			(* cooler type
																			0 = cooler simple version
																			1 = cooler level dependent on valve position
																			2 = cooler level dependent on temperature
																			3 = combined cooler (type 1 and 2) *)
	K_Anz 		:= INT_TO_USINT(LIMIT(1, Para.iEC_NumStages, 16));		(* number cooler stages *)
	Anz_anfhbt	:= INT_TO_USINT(LIMIT(0, Para.iEC_NumDemAux, K_Anz));	(* number cooler stages with demand auxiliaries *)
	K_reg		:= INT_TO_USINT(LIMIT(1, Para.iEC_NumCtr, 11));			(* number controller for y *)
	K_nmp		:= 						 Para.bEC_St1onlyP;				(* selection first stage without fan (only pump)*)
																		(* only IF setting FOR number cooler stages with demand auxiliaries = 0 ! *)
																		(* this option reduces effective cooler fan stages by 1 step ! *)

	(*------------------------------------------------------------------------------------------*)
	(* release emergency cooler from monitoring (from MM_CU) *)
	IN_HC.bEC_Rel;

	(*------------------------------------------------------------------------------------------*)
	(* release for external cooler *)
	OUT_HC.tExCo_Rel.Do	:=	IN_HC.bEng_Aux_Dem_CDR
						AND(bT_HW_Re_Hi OR bT_HW_ReBeEng_Hi);

	(*==========================================================================================*)
	(* emergency cooler control - simple version *)
	IF K_Var = 0 THEN

		OUT_HC.tEC_DemPump.Do	:= (IN_HC.bEC_Rel
								AND IN_HC.bEng_Aux_Dem_CDR AND (bT_AirOutdoor_Hi1 OR NOT Para.bT_AirOutdoor_Active))
								OR IN_HC.tManAuxCtr.bEC_DemPump;	(* Manual operating auxiliaries control - Handbedienebene *)
		OUT_HC.bEmCWP_Dem		:= OUT_HC.tEC_DemPump.Do;

		(* stage 1 *)
		K_ST1	:=  IN_HC.bEC_Rel
				AND	IN_HC.bEng_Aux_Dem_CDR
				AND(bT_AirOutdoor_Hi1 OR NOT Para.bT_AirOutdoor_Active);

		(* stage 2 *)
		K_ST2	:=	IN_HC.bEC_Rel
				AND K_ST1
				AND	IN_HC.bEng_Aux_Dem_CDR
				AND(bT_AirOutdoor_Hi2 OR NOT Para.bT_AirOutdoor_Active);

		(* stage 3 *)
		K_ST3	:=	IN_HC.bEC_Rel
				AND K_ST2
				AND((IN_HC.bEng_Aux_Dem_CDR AND bT_AirOutdoor_Hi3) OR (bT_ECW_Hi1 AND NOT Para.bT_AirOutdoor_Active));

		(* stage 4 *)
		K_ST4	:=	IN_HC.bEC_Rel
				AND K_ST3
				AND((IN_HC.bEng_Aux_Dem_CDR AND bT_AirOutdoor_Hi4) OR (bT_ECW_Hi2 AND NOT Para.bT_AirOutdoor_Active));

	END_IF;

	(*==========================================================================================*)
	(* emergency cooler control - stepper version *)

	IF K_Var > 0 THEN
	(* cooler stages ON/OFF (cooler type 2/3)*)
		bEC_Up   :=     bT_ECW_Hi2 OR      bT_Ch_Hi2 OR      bT_EO_Hi2;
		bEC_Down := NOT bT_ECW_Hi1 AND NOT bT_Ch_Hi1 AND NOT bT_EO_Hi1;

		(*---------------------------------------------------------------------------------------*)
		FA_INIT_0.Word	:=	INT_TO_UINT(K_Var);
		FA_INIT_0;
		K_vent			:=	FA_INIT_0.Bit00;
		K_temp			:=	FA_INIT_0.Bit01;
		muell			:=	FA_INIT_0.Bit02;
		muell			:=	FA_INIT_0.Bit03;
		muell			:=	FA_INIT_0.Bit04;
		muell			:=	FA_INIT_0.Bit05;
		muell			:=	FA_INIT_0.Bit06;
		muell			:=	FA_INIT_0.Bit07;
		muell			:=	FA_INIT_0.Bit08;
		muell			:=	FA_INIT_0.Bit09;
		muell			:=	FA_INIT_0.Bit10;
		muell			:=	FA_INIT_0.Bit11;
		muell			:=	FA_INIT_0.Bit12;
		muell			:=	FA_INIT_0.Bit13;
		muell			:=	FA_INIT_0.Bit14;
		muell			:=	FA_INIT_0.Bit15;

		IF	K_vent AND K_temp	THEN
			Kombi_K		:=	1;
		ELSE
			Kombi_K		:=	0;
		END_IF;

		IF	Anz_anfhbt > 0	THEN
			K_nmp		:=	0;
			K_anfhbt	:=	1;
		ELSE
			K_anfhbt	:=	0;
		END_IF;

		FOR	i			:=	1 TO 16 BY 1 DO
			anfhbt[i]	:=	0;
		END_FOR;
		FOR	i			:=	1 TO Anz_anfhbt BY 1 DO
			anfhbt[i]	:=	1;
		END_FOR;

		(* number effective cooler stages *)
		Anz_st			:=	MIN(K_Anz - (MAX(Anz_anfhbt, 1) - 1) + BOOL_TO_USINT(K_nmp), 16);

		zw				:=	1;
		FOR i			:=	1 TO Anz_st BY 1	DO
			zw			:=	zw * 2;
		END_FOR;

		FA_INIT_1.Word	:=	UDINT_TO_UINT(zw - 1);
		FA_INIT_1;
		ST_1			:=	FA_INIT_1.Bit00;
		ST_2			:=	FA_INIT_1.Bit01;
		ST_3			:=	FA_INIT_1.Bit02;
		ST_4			:=	FA_INIT_1.Bit03;
		ST_5			:=	FA_INIT_1.Bit04;
		ST_6			:=	FA_INIT_1.Bit05;
		ST_7			:=	FA_INIT_1.Bit06;
		ST_8			:=	FA_INIT_1.Bit07;
		ST_9			:=	FA_INIT_1.Bit08;
		ST_10			:=	FA_INIT_1.Bit09;
		ST_11			:=	FA_INIT_1.Bit10;
		ST_12			:=	FA_INIT_1.Bit11;
		ST_13			:=	FA_INIT_1.Bit12;
		ST_14			:=	FA_INIT_1.Bit13;
		ST_15			:=	FA_INIT_1.Bit14;
		ST_16			:=	FA_INIT_1.Bit15;

		(* activation cooler stages *)
		Anz_vent		:=	MIN(K_Anz, 16 - BOOL_TO_USINT(K_nmp));

		zw				:=	1;
		FOR	i			:=	1 TO Anz_vent BY 1	DO
			zw			:=	zw * 2;
		END_FOR;

		FA_INIT_2.Word	:=	UDINT_TO_UINT(zw - 1);
		FA_INIT_2;
		K_ST_1			:=	FA_INIT_2.Bit00;
		K_ST_2			:=	FA_INIT_2.Bit01;
		K_ST_3			:=	FA_INIT_2.Bit02;
		K_ST_4			:=	FA_INIT_2.Bit03;
		K_ST_5			:=	FA_INIT_2.Bit04;
		K_ST_6			:=	FA_INIT_2.Bit05;
		K_ST_7			:=	FA_INIT_2.Bit06;
		K_ST_8			:=	FA_INIT_2.Bit07;
		K_ST_9			:=	FA_INIT_2.Bit08;
		K_ST_10			:=	FA_INIT_2.Bit09;
		K_ST_11			:=	FA_INIT_2.Bit10;
		K_ST_12			:=	FA_INIT_2.Bit11;
		K_ST_13			:=	FA_INIT_2.Bit12;
		K_ST_14			:=	FA_INIT_2.Bit13;
		K_ST_15			:=	FA_INIT_2.Bit14;
		K_ST_16			:=	FA_INIT_2.Bit15;

		(* 3-way cooler valve *)
		CASE K_reg OF							(* selection plant ctr # for 3-way valve (1-11) (cooler type 1/3) *)
		1:	F_SPSR		:=	IN_HC.tCtr_Cust1_In.enable;	(* 1-8 = custom plant ctr - device temperature *)
			rValvePos	:=	IN_HC.tCtr_Cust1_Out.Y;
			REG_INVERT	:=	Para.tCtr_Cust1.invert;
		2:	F_SPSR		:=	IN_HC.tCtr_Cust2_In.enable;
			rValvePos	:=	IN_HC.tCtr_Cust2_Out.Y;
			REG_INVERT	:=	Para.tCtr_Cust2.invert;
		3:	F_SPSR		:=	IN_HC.tCtr_Cust3_In.enable;
			rValvePos	:=	IN_HC.tCtr_Cust3_Out.Y;
			REG_INVERT	:=	Para.tCtr_Cust3.invert;
		4:	F_SPSR		:=	IN_HC.tCtr_Cust4_In.enable;
			rValvePos	:=	IN_HC.tCtr_Cust4_Out.Y;
			REG_INVERT	:=	Para.tCtr_Cust4.invert;
		5:	F_SPSR		:=	IN_HC.tCtr_Cust5_In.enable;
			rValvePos	:=	IN_HC.tCtr_Cust5_Out.Y;
			REG_INVERT	:=	Para.tCtr_Cust5.invert;
		6:	F_SPSR		:=	IN_HC.tCtr_Cust6_In.enable;
			rValvePos	:=	IN_HC.tCtr_Cust6_Out.Y;
			REG_INVERT	:=	Para.tCtr_Cust6.invert;
		7:	F_SPSR		:=	IN_HC.tCtr_Cust7_In.enable;
			rValvePos	:=	IN_HC.tCtr_Cust7_Out.Y;
			REG_INVERT	:=	Para.tCtr_Cust7.invert;
		8:	F_SPSR		:=	IN_HC.tCtr_Cust8_In.enable;
			rValvePos	:=	IN_HC.tCtr_Cust8_Out.Y;
			REG_INVERT	:=	Para.tCtr_Cust8.invert;
		9:	F_SPSR		:=	tCtr_ChC_In.enable;			(* 9   = charge temperature controller *)
			rValvePos	:=	tCtr_ChC_Out.Y;
			REG_INVERT	:=	Para.tCtr_ChC.invert;
		10:	F_SPSR		:=	tCtr_HWRe_In.enable;		(* 10  =  heat water return temperature controller *)
			rValvePos	:=	tCtr_HWRe_Out.Y;
			REG_INVERT	:=	Para.tCtr_HWRe.invert;
		11:	F_SPSR		:=	tCtr_EC_In.enable;			(* 11  =  heat water return temperature after cooler controller *)
			rValvePos	:=	tCtr_EC_Out.Y;
			REG_INVERT	:=	Para.tCtr_EC.invert;
		ELSE
			F_SPSR		:=	FALSE;
			rValvePos	:=	0.0;
			REG_INVERT	:=	FALSE;
		END_CASE;

		IF	NOT REG_INVERT	THEN
			rValvePos	:=	1.0 - rValvePos;
		END_IF;

	    (*---------------------------------------------------------------------------*)
		(* cooler ON *)
		xGRMax_Ventpos5(Gw:= Para.rEC_ValPosLimHi_On, Hy:= Para.rEC_ValPosHyHi_On, In:= rValvePos);

	    (*---------------------------------------------------------------------------*)
		xTOF_K_AUS.IN	:= (K_vent AND xGRMax_Ventpos5.Q AND IN_HC.tPB2MM.bParaSetupOk AND USINT_TO_BOOL(F_SPSR))
						OR (K_temp AND ((bEC_Up OR K_EIN AND NOT bEC_Down) OR K_EIN AND M_KV2));
		xTOF_K_AUS.PT	:=	Para.tiEC_DelayOff;
		xTOF_K_AUS;

		K_EIN			:=	(xTOF_K_AUS.Q OR K_anfhbt) AND IN_HC.bEng_Aux_Dem_CDR AND IN_HC.bEC_Rel;

	    (*---------------------------------------------------------------------------*)
		(* cooler stage plus *)
		xGRMax_Ventpos4(Gw:= Para.rEC_ValPosLimStageUp, Hy:= 0.01, In:= rValvePos);

	    (*---------------------------------------------------------------------------*)
		K_PLUS			:= (K_vent AND xGRMax_Ventpos4.Q AND IN_HC.tPB2MM.bParaSetupOk)
						OR (K_temp AND bEC_Up);

	    (*---------------------------------------------------------------------------*)
		(* cooler stage minus *)
		xGRMin_Ventpos2(Gw:= Para.rEC_ValPosLimStageDown, Hy:= 0.01, In:= rValvePos);

	    (*---------------------------------------------------------------------------*)

		IF	Kombi_K	THEN
			K_MINUS		:= (xGRMin_Ventpos2.Q AND IN_HC.tPB2MM.bParaSetupOk AND bEC_Down) AND NOT K_PLUS;
		ELSE
			K_MINUS		:= (xGRMin_Ventpos2.Q AND IN_HC.tPB2MM.bParaSetupOk AND K_vent OR bEC_Down AND K_temp) AND NOT K_PLUS;
		END_IF;

	    (*---------------------------------------------------------------------------*)
		(* delay between ON *)
		xTOF_PLUS(IN:=	plus, PT:= Para.tiEC_DelayStageUp);
		xR_TRIG_PLUS(CLK:= K_PLUS AND NOT xTOF_PLUS.Q);

	    (*---------------------------------------------------------------------------*)
		(* delay between OFF *)
		xTOF_MINUS(IN:= minus, PT:= Para.tiEC_DelayStageDown);
		xR_TRIG_MINUS(CLK:= K_MINUS AND NOT xTOF_MINUS.Q);

	    (*---------------------------------------------------------------------------*)
		(* reset state maschine *)
		IF	NOT K_EIN	THEN
			schritt		:=	0;
		END_IF;

		(* state maschine *)
		CASE schritt OF	00:	(* cooler stopped *)
			FA_INIT_3.Word	:=	0;
			FA_INIT_3;
			M_KV1			:=	FA_INIT_3.Bit00;
			M_KV2			:=	FA_INIT_3.Bit01;
			M_KV3			:=	FA_INIT_3.Bit02;
			M_KV4			:=	FA_INIT_3.Bit03;
			M_KV5			:=	FA_INIT_3.Bit04;
			M_KV6			:=	FA_INIT_3.Bit05;
			M_KV7			:=	FA_INIT_3.Bit06;
			M_KV8			:=	FA_INIT_3.Bit07;
			M_KV9			:=	FA_INIT_3.Bit08;
			M_KV10			:=	FA_INIT_3.Bit09;
			M_KV11			:=	FA_INIT_3.Bit10;
			M_KV12			:=	FA_INIT_3.Bit11;
			M_KV13			:=	FA_INIT_3.Bit12;
			M_KV14			:=	FA_INIT_3.Bit13;
			M_KV15			:=	FA_INIT_3.Bit14;
			M_KV16			:=	FA_INIT_3.Bit15;

			(* ON 1.stage *)
			IF	K_EIN	THEN
				schritt		:=	10;
			END_IF;

		10:	(* cooler stage 1 *)
			M_KV1			:=	1;
			M_KV2			:=	0;
			(* ON 2.stage *)
			IF	K_PLUS AND (   (K_temp AND bEC_Up AND xR_TRIG_PLUS.Q)
						    OR (K_vent AND xGRMax_Ventpos4.Q)) THEN
				schritt		:=	20;
			END_IF;

		20:	(* cooler stage 2 *)
			M_KV2			:=	1;
			M_KV3			:=	0;
			(* ON 3.stage *)
			IF	K_PLUS AND xR_TRIG_PLUS.Q AND ST_3 THEN
				schritt		:=	30;
			END_IF;
			(* OFF 3.stage *)
			IF	K_MINUS AND (xR_TRIG_MINUS.Q OR NOT ST_3) THEN
				schritt		:=	10;
			END_IF;

		30:	(* cooler stage 3 *)
			M_KV3			:=	1;
			M_KV4			:=	0;
			(* ON 4.stage *)
			IF	K_PLUS AND xR_TRIG_PLUS.Q AND ST_4 THEN
				schritt		:=	40;
			END_IF;
			(* OFF 3.stage *)
			IF	K_MINUS AND (xR_TRIG_MINUS.Q OR NOT ST_4) THEN
				schritt		:=	20;
			END_IF;

		40:	(* cooler stage 4 *)
			M_KV4			:=	1;
			M_KV5			:=	0;
			(* ON 5.stage *)
			IF	K_PLUS AND xR_TRIG_PLUS.Q AND ST_5 THEN
				schritt		:=	50;
			END_IF;
			(* OFF 4.stage *)
			IF	K_MINUS AND (xR_TRIG_MINUS.Q OR NOT ST_5) THEN
				schritt		:=	30;
			END_IF;

		50:	(* cooler stage 5 *)
			M_KV5			:=	1;
			M_KV6			:=	0;
			(* ON 6.stage *)
			IF	K_PLUS AND xR_TRIG_PLUS.Q AND ST_6 THEN
				schritt		:=	60;
			END_IF;
			(* OFF 5.stage *)
			IF	K_MINUS AND (xR_TRIG_MINUS.Q OR NOT ST_6) THEN
				schritt		:=	40;
			END_IF;

		60:	(* cooler stage 6 *)
			M_KV6			:=	1;
			M_KV7			:=	0;
			(* ON 7.stage *)
			IF	K_PLUS AND xR_TRIG_PLUS.Q AND ST_7 THEN
				schritt		:=	70;
			END_IF;
			(* OFF 6.stage *)
			IF	K_MINUS AND (xR_TRIG_MINUS.Q OR NOT ST_7) THEN
				schritt		:=	50;
			END_IF;

		70:	(* cooler stage 7 *)
			M_KV7			:=	1;
			M_KV8			:=	0;
			(* ON 8.stage *)
			IF	K_PLUS AND xR_TRIG_PLUS.Q AND ST_8 THEN
				schritt		:=	80;
			END_IF;
			(* OFF 7.stage *)
			IF	K_MINUS AND (xR_TRIG_MINUS.Q OR NOT ST_8) THEN
				schritt		:=	60;
			END_IF;

		80:	(* cooler stage 8 *)
			M_KV8			:=	1;
			M_KV9			:=	0;
			(* ON 9.stage *)
			IF	K_PLUS AND xR_TRIG_PLUS.Q AND ST_9 THEN
				schritt		:=	90;
			END_IF;
			(* OFF 8.stage *)
			IF	K_MINUS AND (xR_TRIG_MINUS.Q OR NOT ST_9) THEN
				schritt		:=	70;
			END_IF;

		90:	(* cooler stage 9 *)
			M_KV9			:=	1;
			M_KV10			:=	0;
			(* ON 10.stage *)
			IF	K_PLUS AND xR_TRIG_PLUS.Q AND ST_10 THEN
				schritt		:=	100;
			END_IF;
			(* OFF 9.stage *)
			IF	K_MINUS AND (xR_TRIG_MINUS.Q OR NOT ST_10) THEN
				schritt		:=	80;
			END_IF;

		100:(* cooler stage 10 *)
			M_KV10			:=	1;
			M_KV11			:=	0;
			(* ON 11.stage *)
			IF	K_PLUS AND xR_TRIG_PLUS.Q AND ST_11 THEN
				schritt		:=	110;
			END_IF;
			(* OFF 10.stage *)
			IF	K_MINUS AND (xR_TRIG_MINUS.Q OR NOT ST_11) THEN
				schritt		:=	90;
			END_IF;

		110:(* cooler stage 11 *)
			M_KV11			:=	1;
			M_KV12			:=	0;
			(* ON 12.stage *)
			IF	K_PLUS AND xR_TRIG_PLUS.Q AND ST_12 THEN
				schritt		:=	120;
			END_IF;
			(* OFF 11.stage *)
			IF	K_MINUS AND (xR_TRIG_MINUS.Q OR NOT ST_12) THEN
				schritt		:=	100;
			END_IF;

		120:(* cooler stage 12 *)
			M_KV12			:=	1;
			M_KV13			:=	0;
			(* ON 13.stage *)
			IF	K_PLUS AND xR_TRIG_PLUS.Q AND ST_13 THEN
				schritt		:=	130;
			END_IF;
			(* OFF 12.stage *)
			IF	K_MINUS AND (xR_TRIG_MINUS.Q OR NOT ST_13) THEN
				schritt		:=	110;
			END_IF;

		130:(* cooler stage 13 *)
			M_KV13			:=	1;
			M_KV14			:=	0;
			(* ON 14.stage *)
			IF	K_PLUS AND xR_TRIG_PLUS.Q AND ST_14 THEN
				schritt		:=	140;
			END_IF;
			(* OFF 13.stage *)
			IF	K_MINUS AND (xR_TRIG_MINUS.Q OR NOT ST_14) THEN
				schritt		:=	120;
			END_IF;

		140:(* cooler stage 14 *)
			M_KV14			:=	1;
			M_KV15			:=	0;
			(* ON 15.stage *)
			IF	K_PLUS AND xR_TRIG_PLUS.Q AND ST_15 THEN
				schritt		:=	150;
			END_IF;
			(* OFF 14.stage *)
			IF	K_MINUS AND (xR_TRIG_MINUS.Q OR NOT ST_15) THEN
				schritt		:=	130;
			END_IF;

		150:(* cooler stage 15 *)
			M_KV15			:=	1;
			M_KV16			:=	0;
			(* ON 16.stage *)
			IF	K_PLUS AND xR_TRIG_PLUS.Q AND ST_16 THEN
				schritt		:=	160;
			END_IF;
			(* OFF 15.stage *)
			IF	K_MINUS AND (xR_TRIG_MINUS.Q OR NOT ST_16) THEN
				schritt		:=	140;
			END_IF;

		160:(* cooler stage 16 *)
			M_KV16			:=	1;
			(* OFF 16.stage *)
			IF	K_MINUS	THEN
				schritt		:=	150;
			END_IF;
		END_CASE;

		(* dump radiator pump *)
		OUT_HC.tEC_DemPump.Do	:= (IN_HC.bEng_Aux_Dem_CDR AND(((M_KV1  OR  xGRMax_Ventpos5.Q)AND NOT Kombi_K)
															  OR(M_KV1  AND xGRMax_Ventpos5.Q)))
								 OR IN_HC.tManAuxCtr.bEC_DemPump;	(* Manual operating auxiliaries control - Handbedienebene *)
		OUT_HC.bEmCWP_Dem		:= OUT_HC.tEC_DemPump.Do;

		(* connection steps to sequencing *)
		K_ST1	:= (xGRMax_Ventpos5.Q	OR 	NOT Kombi_K)
				AND(   (M_KV1  	AND NOT K_nmp)
					OR	M_KV2);

		K_ST2	:= (xGRMax_Ventpos5.Q 	OR 	NOT Kombi_K)
				AND(   (M_KV1  	AND 	anfhbt[2])
					OR (M_KV2  	AND NOT K_nmp)
					OR	M_KV3);

		K_ST3	:= (xGRMax_Ventpos5.Q	OR 	NOT Kombi_K)
				AND(   (M_KV1  	AND 	anfhbt[3])
					OR (M_KV2  	AND 	anfhbt[2])
					OR (M_KV3  	AND NOT K_nmp)
					OR	M_KV4);

		K_ST4	:= (xGRMax_Ventpos5.Q	OR 	NOT Kombi_K)
				AND(   (M_KV1  	AND 	anfhbt[4])
					OR (M_KV2  	AND 	anfhbt[3])
					OR (M_KV3  	AND 	anfhbt[2])
					OR (M_KV4  	AND NOT K_nmp)
					OR	M_KV5);

		K_ST5	:= (xGRMax_Ventpos5.Q 	OR 	NOT Kombi_K)
				AND(   (M_KV1  	AND 	anfhbt[5])
					OR (M_KV2  	AND 	anfhbt[4])
					OR (M_KV3  	AND 	anfhbt[3])
					OR (M_KV4  	AND 	anfhbt[2])
					OR (M_KV5  	AND NOT K_nmp)
					OR	M_KV6);

		K_ST6	:= (xGRMax_Ventpos5.Q 	OR 	NOT Kombi_K)
				AND(   (M_KV1	AND 	anfhbt[6])
					OR (M_KV2  	AND 	anfhbt[5])
					OR (M_KV3  	AND 	anfhbt[4])
					OR (M_KV4  	AND 	anfhbt[3])
					OR (M_KV5  	AND 	anfhbt[2])
					OR (M_KV6  	AND NOT K_nmp)
					OR  M_KV7);

		K_ST7	:= (xGRMax_Ventpos5.Q 	OR 	NOT Kombi_K)
				AND(   (M_KV1  	AND 	anfhbt[7])
					OR (M_KV2  	AND 	anfhbt[6])
					OR (M_KV3  	AND 	anfhbt[5])
					OR (M_KV4  	AND 	anfhbt[4])
					OR (M_KV5  	AND 	anfhbt[3])
					OR (M_KV6  	AND 	anfhbt[2])
					OR (M_KV7  	AND NOT K_nmp)
					OR  M_KV8);

		K_ST8	:= (xGRMax_Ventpos5.Q 	OR 	NOT Kombi_K)
				AND(   (M_KV1  	AND 	anfhbt[8])
					OR (M_KV2  	AND 	anfhbt[7])
					OR (M_KV3  	AND 	anfhbt[6])
					OR (M_KV4  	AND 	anfhbt[5])
					OR (M_KV5  	AND 	anfhbt[4])
					OR (M_KV6  	AND 	anfhbt[3])
					OR (M_KV7  	AND 	anfhbt[2])
					OR (M_KV8  	AND NOT K_nmp)
					OR  M_KV9);

		K_ST9	:= (xGRMax_Ventpos5.Q 	OR 	NOT Kombi_K)
				AND(   (M_KV1  	AND 	anfhbt[9])
					OR (M_KV2  	AND 	anfhbt[8])
					OR (M_KV3  	AND 	anfhbt[7])
					OR (M_KV4  	AND 	anfhbt[6])
					OR (M_KV5  	AND 	anfhbt[5])
					OR (M_KV6  	AND 	anfhbt[4])
					OR (M_KV7  	AND 	anfhbt[3])
					OR (M_KV8  	AND 	anfhbt[2])
					OR (M_KV9  	AND NOT K_nmp)
					OR  M_KV10);

		K_ST10	:= (xGRMax_Ventpos5.Q 	OR 	NOT Kombi_K)
				AND(   (M_KV1  	AND 	anfhbt[10])
					OR (M_KV2  	AND 	anfhbt[9])
					OR (M_KV3  	AND 	anfhbt[8])
					OR (M_KV4  	AND 	anfhbt[7])
					OR (M_KV5  	AND 	anfhbt[6])
					OR (M_KV6  	AND 	anfhbt[5])
					OR (M_KV7  	AND 	anfhbt[4])
					OR (M_KV8  	AND 	anfhbt[3])
					OR (M_KV9  	AND 	anfhbt[2])
					OR (M_KV10 	AND NOT K_nmp)
					OR  M_KV11);

		K_ST11	:= (xGRMax_Ventpos5.Q 	OR 	NOT Kombi_K)
				AND(   (M_KV1  	AND 	anfhbt[11])
					OR (M_KV2  	AND 	anfhbt[10])
					OR (M_KV3  	AND 	anfhbt[9])
					OR (M_KV4  	AND 	anfhbt[8])
					OR (M_KV5  	AND 	anfhbt[7])
					OR (M_KV6  	AND 	anfhbt[6])
					OR (M_KV7  	AND 	anfhbt[5])
					OR (M_KV8  	AND 	anfhbt[4])
					OR (M_KV9  	AND 	anfhbt[3])
					OR (M_KV10 	AND 	anfhbt[2])
					OR (M_KV11 	AND NOT K_nmp)
					OR  M_KV12);

		K_ST12	:= (xGRMax_Ventpos5.Q 	OR 	NOT Kombi_K)
				AND(   (M_KV1  	AND 	anfhbt[12])
					OR (M_KV2  	AND 	anfhbt[11])
					OR (M_KV3  	AND 	anfhbt[10])
					OR (M_KV4  	AND 	anfhbt[9])
					OR (M_KV5  	AND 	anfhbt[8])
					OR (M_KV6  	AND 	anfhbt[7])
					OR (M_KV7  	AND 	anfhbt[6])
					OR (M_KV8  	AND 	anfhbt[5])
					OR (M_KV9  	AND 	anfhbt[4])
					OR (M_KV10 	AND 	anfhbt[3])
					OR (M_KV11 	AND 	anfhbt[2])
					OR (M_KV12 	AND NOT K_nmp)
					OR  M_KV13);

		K_ST13	:= (xGRMax_Ventpos5.Q 	OR 	NOT Kombi_K)
				AND(   (M_KV1  	AND 	anfhbt[13])
					OR (M_KV2  	AND 	anfhbt[12])
					OR (M_KV3  	AND 	anfhbt[11])
					OR (M_KV4  	AND 	anfhbt[10])
					OR (M_KV5  	AND 	anfhbt[9])
					OR (M_KV6  	AND 	anfhbt[8])
					OR (M_KV7  	AND 	anfhbt[7])
					OR (M_KV8  	AND 	anfhbt[6])
					OR (M_KV9  	AND 	anfhbt[5])
					OR (M_KV10 	AND 	anfhbt[4])
					OR (M_KV11 	AND 	anfhbt[3])
					OR (M_KV12 	AND 	anfhbt[2])
					OR (M_KV13 	AND NOT K_nmp)
					OR  M_KV14);

		K_ST14	:= (xGRMax_Ventpos5.Q 	OR 	NOT Kombi_K)
				AND(   (M_KV1  	AND 	anfhbt[14])
					OR (M_KV2  	AND 	anfhbt[13])
					OR (M_KV3  	AND 	anfhbt[12])
					OR (M_KV4  	AND 	anfhbt[11])
					OR (M_KV5  	AND 	anfhbt[10])
					OR (M_KV6  	AND 	anfhbt[9])
					OR (M_KV7  	AND 	anfhbt[8])
					OR (M_KV8  	AND 	anfhbt[7])
					OR (M_KV9  	AND 	anfhbt[6])
					OR (M_KV10 	AND 	anfhbt[5])
					OR (M_KV11 	AND 	anfhbt[4])
					OR (M_KV12 	AND 	anfhbt[3])
					OR (M_KV13 	AND 	anfhbt[2])
					OR (M_KV14 	AND NOT K_nmp)
					OR  M_KV15);

		K_ST15	:= (xGRMax_Ventpos5.Q 	OR 	NOT Kombi_K)
				AND(   (M_KV1  	AND 	anfhbt[15])
					OR (M_KV2  	AND 	anfhbt[14])
					OR (M_KV3  	AND 	anfhbt[13])
					OR (M_KV4  	AND 	anfhbt[12])
					OR (M_KV5  	AND 	anfhbt[11])
					OR (M_KV6  	AND 	anfhbt[10])
					OR (M_KV7  	AND 	anfhbt[9])
					OR (M_KV8  	AND 	anfhbt[8])
					OR (M_KV9  	AND 	anfhbt[7])
					OR (M_KV10 	AND 	anfhbt[6])
					OR (M_KV11 	AND 	anfhbt[5])
					OR (M_KV12 	AND 	anfhbt[4])
					OR (M_KV13 	AND 	anfhbt[3])
					OR (M_KV14 	AND 	anfhbt[2])
					OR (M_KV15 	AND NOT K_nmp)
					OR  M_KV16);

		K_ST16	:= (xGRMax_Ventpos5.Q 	OR 	NOT Kombi_K)
				AND(   (M_KV1  	AND 	anfhbt[16])
					OR (M_KV2  	AND 	anfhbt[15])
					OR (M_KV3  	AND 	anfhbt[14])
					OR (M_KV4  	AND 	anfhbt[13])
					OR (M_KV5  	AND 	anfhbt[12])
					OR (M_KV6  	AND 	anfhbt[11])
					OR (M_KV7  	AND 	anfhbt[10])
					OR (M_KV8  	AND 	anfhbt[9])
					OR (M_KV9  	AND 	anfhbt[8])
					OR (M_KV10 	AND 	anfhbt[7])
					OR (M_KV11 	AND 	anfhbt[6])
					OR (M_KV12 	AND 	anfhbt[5])
					OR (M_KV13 	AND 	anfhbt[4])
					OR (M_KV14 	AND 	anfhbt[3])
					OR (M_KV15 	AND 	anfhbt[2])
					OR (M_KV16 	AND NOT K_nmp));

		(* copy for summation *)
		KST[1]	:=	BOOL_TO_USINT(M_KV1);
		KST[2]	:=	BOOL_TO_USINT(M_KV2);
		KST[3]	:=	BOOL_TO_USINT(M_KV3);
		KST[4]	:=	BOOL_TO_USINT(M_KV4);
		KST[5]	:=	BOOL_TO_USINT(M_KV5);
		KST[6]	:=	BOOL_TO_USINT(M_KV6);
		KST[7]	:=	BOOL_TO_USINT(M_KV7);
		KST[8]	:=	BOOL_TO_USINT(M_KV8);
		KST[9]	:=	BOOL_TO_USINT(M_KV9);
		KST[10]	:=	BOOL_TO_USINT(M_KV10);
		KST[11]	:=	BOOL_TO_USINT(M_KV11);
		KST[12]	:=	BOOL_TO_USINT(M_KV12);
		KST[13]	:=	BOOL_TO_USINT(M_KV13);
		KST[14]	:=	BOOL_TO_USINT(M_KV14);
		KST[15]	:=	BOOL_TO_USINT(M_KV15);
		KST[16]	:=	BOOL_TO_USINT(M_KV16);

		(* ON / OFF cooler stages *)
		summe := 0;
		FOR i:= 1 TO 16 BY 1 DO
			summe := summe + KST[i];
		END_FOR;

		plus := 0;
		IF (summe > summe_old) THEN
			plus :=	1;
		END_IF;

		minus := 0;
		IF (summe < summe_old) THEN
			minus := 1;
		END_IF;

		summe_old := summe;

	END_IF;
	(*------------------------------------------------------------------------------------------*)

END_PROGRAM
```

#### EC.var
```iecst
VAR
	rValvePos : REAL; (*valve position*)
	muell : BOOL := FALSE;
	K_Var : INT; (*emergency cooler variant(Para.iEC_OpMode)*)
	K_Anz : USINT; (*emergency cooler *)
	K_nmp : BOOL; (*1.stage only with pump*)
	K_reg : USINT;
	ST_5 : BOOL;
	ST_4 : BOOL;
	ST_7 : BOOL;
	ST_6 : BOOL;
	ST_3 : BOOL;
	REG_INVERT : BOOL;
	ST_1 : BOOL;
	minus : BOOL := 0;
	plus : BOOL := 0;
	ST_8 : BOOL;
	ST_15 : BOOL;
	ST_14 : BOOL;
	ST_2 : BOOL;
	ST_16 : BOOL;
	ST_13 : BOOL;
	ST_9 : BOOL;
	ST_10 : BOOL;
	ST_11 : BOOL;
	ST_12 : BOOL;
	anfhbt : ARRAY[0..16] OF BOOL;
	xGRMax_Ventpos4 : GR_MAXR;
	xGRMax_Ventpos5 : GR_MAXR;
	xGRMin_Ventpos2 : GR_MINR;
	xR_TRIG_MINUS : R_TRIG;
	xR_TRIG_PLUS : R_TRIG;
	xTOF_MINUS : TOF;
	xTOF_PLUS : TOF;
	xTOF_K_AUS : TOF;
	zw : UDINT;
	Anz_st : USINT;
	summe : USINT;
	summe_old : USINT := 0;
	schritt : USINT := 0;
	i : USINT;
	F_SPSR : USINT;
	Anz_vent : USINT;
	KST : ARRAY[0..16] OF USINT;
	FA_INIT_0 : WDtoBIT;
	FA_INIT_1 : WDtoBIT;
	FA_INIT_2 : WDtoBIT;
	FA_INIT_3 : WDtoBIT;
END_VAR
```

### Program Logical/HeatingCooling/ChC (IEC, version 4.07.0) - charge cooler
